KUKA KRL program: kuka_pick_and_place.src

&ACCESS RVP
&REL 1
&PARAM TEMPLATE = C:\KRC\Roboter\Template
&PARAM EDITMASK = *
DEF PICK_PLACE( )
;FOLD INI
  BAS (#INITMOV,0 )
;ENDFOLD
PTP  HOME
LIN  P_PICK_APPR
LIN  P_PICK
; (Close gripper - external IO call placeholder)
LIN  P_PICK_APPR
PTP  P_PLACE_APPR
LIN  P_PLACE
; (Open gripper - external IO call placeholder)
LIN  P_PLACE_APPR
PTP  HOME
END
